DATA_BLOCK "DB_RobotMissionStatus"
{ S7_Optimized_Access := 'TRUE' }
VERSION : 0.1
NON_RETAIN
"Robot_mission_STATUS"

BEGIN

END_DATA_BLOCK

